RoboDK station: assembly.rdk

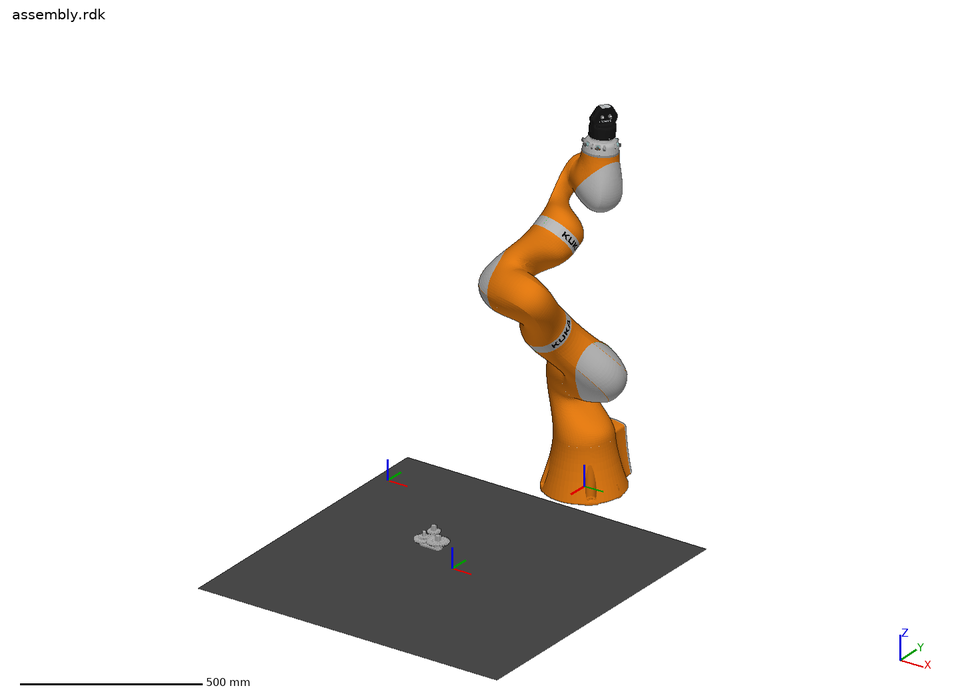
[picture v0: the station drawn from its stored meshes, robots at their saved joint values, targets as dots, program paths as lines]
Station assembly (saved by RoboDK 5.2.1). Poses are relative to the parent item; angles as X-Y-Z fixed-axis rotations.
Station parameters (name, value as stored): AutoAvoidance, YuMi IRB 14000-0.5/0.5-R, AutoAvoidance-Rob YuMi IRB 14000-0.5/0.5-R
  - frame workspace at (0, 0, 200) mm
    - object assembly_place at (0, 0, 0) mm, size 1000 x 1000 x 0.5 mm, geometry from plane_1m.sld
      - object base_plate at (-150, 80, 0) mm, size 71.4 x 71.9 x 41 mm, geometry from base_plate.stl
      - object compound_gear at (-150, 80, 15) mm, size 60.6 x 60.6 x 11.4 mm, geometry from compound_gear.stl
      - object shaft1 at (-150, 126, 41) mm, rotated rx 180 ry 0 rz 180 deg, size 12 x 12 x 38.5 mm, geometry from shaft1.stl
      - object shaft2 at (-104, 80, 41) mm, rotated rx 180 ry 0 rz -180 deg, size 14 x 14 x 38.5 mm, geometry from shaft2.stl
      - object gear1 at (-150, 126, 20) mm, size 39.6 x 39.4 x 5.4 mm, geometry from gear1.stl
      - object gear2 at (-104, 80, 20) mm, size 64.9 x 64.9 x 5.4 mm, geometry from gear2.stl
  - frame KUKA LBR iiwa 14 R820 Base at (0, 630, 200) mm, rotated rx 0 ry 0 rz -90 deg
    - robot robot (model KUKA LBR iiwa 14 R820): 7 axes, payload 14 kg, reach 820 mm, repeatability 0.1 mm, weight 29.9 kg
        modified DH rows (alpha deg, a mm, theta deg, d mm): 0, 0, 0, 360; -90, 0, 0, 0; 90, 0, 0, 420; -90, 0, 0, 0; 90, 0, 0, 400; -90, 0, 0, 0; 90, 0, 0, 126
        joint limits [-170, -120, -170, -120, -170, -120, -175] to [170, 120, 170, 120, 170, 120, 175]; home [0, 0, 0, -90, 0, 0, 0]; saved at [-10.708, 40, 0, -93.578, 0, 46.422, 169.292]
      - robot RobotiQ 2F85: 1 axes, payload 5 kg
          joint limits [0] to [85]; home [85]; saved at [19.65]
      - tool tcp, TCP at (0, 0, 100) mm
  - frame parts_ref at (-460, 350, 200) mm
  - Python program run_assembly (listed below)

--- Python program run_assembly ---
"""All in One RoboDK script"""
from abc import ABC, abstractmethod
import robolink
import json
import robodk
import numpy as np


class RDKSimulation(ABC):
    """RoboDK simulation class."""
    def __init__(self):
        self.rblink = robolink.Robolink()
        self.simulation_speed = 1
        self.refresh_rate = 0.005

    @abstractmethod
    def run(self):
        """Runs simulation."""
        raise NotImplementedError(f'You have to implement this method!')

    @abstractmethod
    def reset(self):
        """Resets simulation."""
        raise NotImplementedError('You have to implement this method!')


class PickablePart:
    """Item class."""

    def __init__(self,
                 item,
                 part_id,
                 pick_approach_pose_offset,
                 pick_pose_offset,
                 pick_retract_offset,
                 place_approach_pose_offset,
                 place_pose_offset,
                 place_retract_offset):
        self.item = item
        self.part_id = part_id
        self.pick_approach_pose_offset = pick_approach_pose_offset
        self.pick_pose_offset = pick_pose_offset
        self.pick_retract_pose_offset = pick_retract_offset
        self.place_approach_pose_offset = place_approach_pose_offset
        self.place_pose_offset = place_pose_offset
        self.place_retract_pose_offset = place_retract_offset


class Assembly(RDKSimulation):
    """Assembly of parts."""

    def __init__(self, recipe):
        super().__init__()

        # set simulation speed
        self.rblink.setSimulationSpeed(1)

        # get robot
        self.robot = self.rblink.Item('robot')
        # wrt to the station, useful for calculating positions
        self.rinv = robodk.invH(self.robot.PoseAbs())

        # TCP
        self.tcp = self.rblink.Item('tcp')

        # assembly place like table
        self.assembly_place = self.rblink.Item('assembly_place')
        # target assembly pose in robot reference frame
        self.target_pos3d = np.array([550, -150, 0])  # should be checked for the reachability

        # initial assembly parts position
        self.parts_ref = self.rblink.Item('parts_ref')

        # read recipe
        self.assembly_sequence = recipe['sequence']
        self.parts = {}
        for part_data in recipe['parts']:
            part_id = part_data['part_id']
            self.parts[part_id] = PickablePart(item=self.rblink.Item(part_id),
                                               part_id=part_id,
                                               pick_approach_pose_offset=part_data['pick_approach_pose_offset'],
                                               pick_pose_offset=part_data['pick_pose_offset'],
                                               pick_retract_offset=part_data['pick_retract_pose_offset'],
                                               place_approach_pose_offset=part_data['place_approach_pose_offset'],
                                               place_pose_offset=part_data['place_pose_offset'],
                                               place_retract_offset=part_data['place_retract_pose_offset'])

        # this is fixed for now
        self.initial_poses = {
            'base_plate': [0, 60, 0, 0, 0, 0],
            'compound_gear': [0, -30, 0, 0, 0, 0],
            'gear1': [0, -120, 0, 0, 0, 0],
            'gear2': [90, -160, 0, 0, 0, 0],
            'shaft1': [100, 0, 39, 0, -180, 0],
            'shaft2': [100, -70, 39, 0, -180, 0]
        }

        self.reset()

    def run(self):
        """Runs simulation."""
        # target_pose = robodk.Pose(550, -70, 0, 0, 0, 0)
        # self.pick_and_place(item, target_pose)
        self.assemble()

    def move_robot(self, pos3d, offset):
        """Moves robot to the 3d position with given offset."""
        pose = robodk.Pose(*(np.array([*pos3d, 0, 0, 0]) + offset))
        self.robot.MoveJ(pose)

    def assemble(self):
        """Assemble the parts in the sequence."""
        for part_id in self.assembly_sequence:
            part = self.parts[part_id]
            self.pick_and_place(part)

    def pick_and_place(self, part):
        """Picks and places the part."""
        part_pos3d = (self.rinv * part.item.PoseAbs()).Pos()

        # 1. Go to the pick approach pose.
        self.move_robot(part_pos3d, part.pick_approach_pose_offset)

        # 2. Go to the pick pose.
        self.move_robot(part_pos3d, part.pick_pose_offset)

        # 3. Pick the part.
        part.item.setParentStatic(self.tcp)

        # 4. Go to the pick retract pose.
        self.move_robot(part_pos3d, part.pick_retract_pose_offset)

        # 5. Go to the place approach pose.
        self.move_robot(self.target_pos3d, part.place_approach_pose_offset)

        # 6. Go to the place pose.
        self.move_robot(self.target_pos3d, part.place_pose_offset)

        # 7. Place the part.
        part.item.setParentStatic(self.assembly_place)

        # 8. Go to the place retract pose.
        self.move_robot(self.target_pos3d, part.place_retract_pose_offset)

    def reset(self):
        """Resets simulation."""

        # reset robot to the home position
        # for KUKA LBR iiwa 14 R820
        self.robot.setJoints([0, 0, 0, -90, 0, 0, 0])

        for part in self.parts.values():
            part.item.setParentStatic(self.parts_ref)
            part.item.setPose(robodk.Pose(*self.initial_poses[part.part_id]))


recipe = """{
  "parts": [
    {
      "part_id": "base_plate",
      "pick_approach_pose_offset": [0, 0, 120, 180, 0, 0],
      "pick_pose_offset": [0, 0, 80, 180, 0, 0],
      "pick_retract_pose_offset": [0, 0, 160, 180, 0, 0],
      "place_approach_pose_offset": [0, 0, 120, 180, 0, 0],
      "place_pose_offset": [0, 0, 80, 180, 0, 0],
      "place_retract_pose_offset": [0, 0, 160, 180, 0, 0]
    },

    {
      "part_id": "compound_gear",
      "pick_approach_pose_offset": [0, 0, 120, 180, 0, 0],
      "pick_pose_offset": [0, 0, 75, 180, 0, 0],
      "pick_retract_pose_offset": [0, 0, 160, 180, 0, 0],
      "place_approach_pose_offset": [0, 0, 140, 180, 0, 0],
      "place_pose_offset": [0, 0, 90, 180, 0, 0],
      "place_retract_pose_offset": [0, 0, 160, 180, 0, 0]
    },

    {
      "part_id": "shaft1",
      "pick_approach_pose_offset": [0, 0, 120, 180, 0, 0],
      "pick_pose_offset": [0, 0, 45, 180, 0, 0],
      "pick_retract_pose_offset": [0, 0, 180, 180, 0, 0],
      "place_approach_pose_offset": [-46, 0, 180, 180, 0, 0],
      "place_pose_offset": [-46, 0, 86, 180, 0, 0],
      "place_retract_pose_offset": [-46, 0, 180, 180, 0, 0]
    },

    {
      "part_id": "shaft2",
      "pick_approach_pose_offset": [0, 0, 120, 180, 0, 0],
      "pick_pose_offset": [0, 0, 45, 180, 0, 0],
      "pick_retract_pose_offset": [0, 0, 180, 180, 0, 0],
      "place_approach_pose_offset": [0, 46, 140, 180, 0, 0],
      "place_pose_offset": [0, 46, 86, 180, 0, 0],
      "place_retract_pose_offset": [0, 46, 180, 180, 0, 0]
    },

    {
      "part_id": "gear1",
      "pick_approach_pose_offset": [0, 0, 120, 180, 0, 0],
      "pick_pose_offset": [0, 0, 65, 180, 0, 0],
      "pick_retract_pose_offset": [0, 0, 180, 180, 0, 0],
      "place_approach_pose_offset": [-46, 0, 180, 180, 0, 0],
      "place_pose_offset": [-46, 0, 85, 180, 0, 0],
      "place_retract_pose_offset": [-46, 0, 180, 180, 0, 0]
    },

    {
      "part_id": "gear2",
      "pick_approach_pose_offset": [0, 0, 120, 180, 0, 0],
      "pick_pose_offset": [0, 0, 45, 180, 0, 0],
      "pick_retract_pose_offset": [0, 0, 180, 180, 0, 0],
      "place_approach_pose_offset": [0, 46, 140, 180, 0, 0],
      "place_pose_offset": [0, 46, 65, 180, 0, 0],
      "place_retract_pose_offset": [0, 46, 180, 180, 0, 0]
    }
  ],

  "sequence": [
    "base_plate", "compound_gear", "shaft1", "shaft2", "gear1", "gear2"
  ]
}"""

if __name__ == '__main__':
    assembly_recipe = json.loads(recipe)
    sim = Assembly(assembly_recipe)
    sim.run()
